FUNCTION_BLOCK TOffTimer
VAR
    TOF1 : TOF;
END_VAR

METHOD Delay : BOOL
VAR_INPUT
    In : BOOL;
END_VAR
TOF1(IN := In);
Delay := TOF1.Q;
END_METHOD

METHOD FB_init : BOOL
VAR_INPUT
	bInitRetains : BOOL; // if TRUE, the retain variables are initialized (warm start / cold start)
	bInCopyCode : BOOL;  // if TRUE, the instance afterwards gets moved into the copy code (online change)
    PresetTime : LREAL; // seconds
END_VAR
TOF1.PT := LREAL_TO_TIME(PresetTime * 1000);
END_METHOD

PROPERTY OutputState : BOOL
GET
OutputState := TOF1.Q;
END_GET
END_PROPERTY

PROPERTY PresetTime : LREAL
GET
PresetTime := TIME_TO_LREAL(TOF1.PT)/1000.0; // in seconds
END_GET
SET
TOF1.PT := LREAL_TO_TIME(PresetTime * 1000);
END_SET
END_PROPERTY

END_FUNCTION_BLOCK

(* stored: Version 1.1.0.1, ProductVersion 3.1.4024.3
   POU TOffTimer: Id {41674d6f-3be8-0a43-194c-c209f1d77075}, SpecialFunc None
   Method Delay: Id {e4015604-15d0-0b2e-0c9b-4e327928efa4}
   Method FB_init: Id {3a611803-2504-026b-2a66-962e6c3f8665}
   Property OutputState: Id {6e266f24-8214-0bb2-019b-00c12bc3c072}
   Get Get: Id {46336c7a-d2de-0080-14ca-9dc2d99ba2f2}
   Property PresetTime: Id {8dc3a5ed-30c1-033d-1873-570fcf6b7ad7}
   Get Get: Id {0bfc87d1-4ceb-0168-10ae-c4604a854bd4}
   Set Set: Id {51db4b2c-86c4-0f9c-0244-4af693f05f93} *)
